Fanuc KAREL source: kb00076.KL

-- PROVISIONAL review KL for V770-1; original PC SHA256 f91a445edfeb9c2137934b770fc54e181e6bda922a8fbe32fa757bd74d0e86ec
-- Incomplete behavior may be omitted. Consult companion uncertainty JSON. Do not deploy.
PROGRAM KB00076
%NOLOCKGROUP
-- UNRESOLVED_DECL P1 type=000101
-- UNRESOLVED_DECL P2 type=000101
-- UNRESOLVED_DECL P3 type=000101
-- UNRESOLVED_DECL RESULT type=000101
BEGIN
  -- UNRESOLVED_PC offsets 5-56; opcodes 27,22,1C,22,1C,22,1C,76,7E,4A
  -- UNRESOLVED_PC offsets 61-65; opcodes 7F
END KB00076
